PROGRAM MAIN
VAR
 aTransferLines  : ARRAY[1..3] OF SM_TransferLine;
 fbSymbolPathStorage : SymbolPathStorage;
END_VAR

END_PROGRAM

(* stored: Version 1.1.0.1, ProductVersion 3.1.4024.0
   POU MAIN: Id {c83d4c06-b08c-4f63-b878-b3a4e7399e2e}, SpecialFunc None *)
